// TIA Portal V19 export
DATA_BLOCK "A01_HMI_IDB"   // DB88
AUTHOR : Piemme
FAMILY : System
// stored: InstanceOfName A01_HMI_FB, InstanceOfType FB
"A01_HMI_FB"
   // VAR
   //    MB1_Decoder { ExternalAccessible := 'False'; ExternalVisible := 'False'; ExternalWritable := 'False'} : "ButtonsHMIDecoder";
   // END_VAR
BEGIN
END_DATA_BLOCK
